VISUALIZATION Math  // 1920x1080
END_VISUALIZATION

(* stored: Version 1.1.0.1, ProductVersion 3.1.4024.12
   Visu Math: Id {6e67d57f-c320-4078-8c97-73aac621b48e} *)
